// Mitsubishi GX Works2 project: 22   PLC: FX3G

// task Task_01 (event TRUE, interval 0, priority 31): POU_01

PROGRAM POU_01
VAR
  rate : INT;
  wstep : INT;
  ton1 : TON;
  wtime : TIME;
  counter : INT;
END_VAR
M99 := FALSE AND
M1 AND M2 AND M3 AND
Y1 AND Y2 AND Y3 AND Y4;

IF M8002 THEN
	wstep := 0;
END_IF;

CASE wstep OF
	0:
		zrst(TRUE, Y1, Y4);
		ton1(in := FALSE);
		
		IF M1 THEN
			wtime := t#10s;
			counter := 1;
			Y1 := TRUE;
			wstep := 20;
		END_IF;
		IF M2 THEN
			wstep := 40;
		END_IF;
		IF M3 THEN
			wtime := t#5s;
			counter := 1;
			Y1 := TRUE;
			wstep := 20;
		END_IF;
		
	20:
		ton1(in := NOT ton1.q, pt := wtime);
		IF ton1.q THEN
			Z0 := counter;
			Y0Z0 := FALSE;
			counter := counter + 1;
			Z0 := counter;
			Y0Z0 := TRUE;
		END_IF;
		
		IF counter = 5 THEN
			wstep := 0;
		END_IF;

	40:
		Y4 := TRUE;
		ton1(in := NOT ton1.q, pt := t#10s);
		
		IF ton1.q THEN
			wstep := 0;
		END_IF;

END_CASE;
END_PROGRAM
